(* Logix 5000 project; controller AdvManLab vendor 1 type 14 code 158 rev 28.12; software revision 28.01; part 11 of 13 *)
(* tags used below, declared in another part *)
   RFID_Address : DINT;
   RFID_Length : DINT;
   RFID_Read_1 : BOOL;
   RFID_Read_3 : BOOL;
   RFID_Read_5 : BOOL;
   RFID_Read_Byte_Start_1 : BOOL;
   RFID_Read_Byte_Start_3 : BOOL;
   RFID_Read_Byte_Start_5 : BOOL;
   RFID_Read_InProgress_1 : BOOL;
   RFID_Read_InProgress_3 : BOOL;
   RFID_Read_InProgress_5 : BOOL;
   ABB_Loop_Conv_ES_Ch1 : BOOL;   // Cell 3 Conveyor Pull Cord / E-Stop Ch1
   ABB_Loop_Conv_ES_Ch2 : BOOL;   // Cell 3 Conveyor Pull Cord / E-Stop Ch2
   ABB_Loop_Conv_Safety_OK : BOOL;
   ABBLoopPullCordES : EMERGENCY_STOP;   // EStop / Cable On ABB Loop
   ABBLoopSTO_O1 : BOOL;
   ABBLoopSTO_O2 : BOOL;
   ASynch : BOOL;
   AutoProgStart : TIMER;
   C1_Robot_ES_OK : BOOL;
   C1_Robot_Gates_OK : BOOL;
   C1S : Fanuc_Cell_Safe;
   C2_Robot_ES_OK : BOOL;
   C2_Robot_Gates_OK : BOOL;
   C2S : Fanuc_Cell_Safe;
   C3_Robot_ES_OK : BOOL;
   C3_Robot_Gates_OK : BOOL;
   C3S : ABB_Cell_Safe;
   Cell1EntryLC : LIGHT_CURTAIN;   // Cell 1 Conveyor Entry Light Screen
   Cell1EntryLCMute : MUTING_TWO_SENSOR_SYM;   // Celll 1 Entry LC Muting
   Cell1ExitLC : LIGHT_CURTAIN;   // Cell 1 Conveyor Exit Light Screen
   Cell1ExitLCMute : MUTING_TWO_SENSOR_SYM;   // Celll 1 Exit LC Muting
   Cell1GateSW : REDUNDANT_INPUT;   // Cell 1 Entry Gate Switch
   Cell2EntryLC : LIGHT_CURTAIN;   // Cell 2 Conveyor Entry Light Screen
   Cell2EntryLCMute : MUTING_TWO_SENSOR_SYM;   // Celll 2 Entry LC Muting
   Cell2ExitLC : LIGHT_CURTAIN;   // Cell 2 Conveyor Exit Light Screen
   Cell2ExitLCMute : MUTING_TWO_SENSOR_SYM;   // Celll 2 Exit LC Muting
   Cell2GateSW : REDUNDANT_INPUT;   // Cell 2 Entry Gate Switch
   Cell3EntryLC : LIGHT_CURTAIN;   // Cell 3 Conveyor Entry Light Screen
   Cell3EntryLCMute : MUTING_TWO_SENSOR_SYM;   // Celll 3 Entry LC Muting
   Cell3ExitLC : LIGHT_CURTAIN;   // Cell 3 Conveyor Exit Light Screen
   Cell3ExitLCMute : MUTING_TWO_SENSOR_SYM;   // Celll 3 Exit LC Muting
   Cell3GateSW : REDUNDANT_INPUT;   // Cell 3 Entry Gate Switch
   Cell_1 : Fanuc_Cell;
   Cell_2 : Fanuc_Cell;
   CircuitResetSafe : BOOL;   // Signal to Reset Circuits
   CNC1_Door : REDUNDANT_INPUT;   // CNC1 Door Switch
   CNC1_EStop : EMERGENCY_STOP;
   CNC1_LC : LIGHT_CURTAIN;   // CNC1 to Cell 1 Light Screen
   CNC2_Door : REDUNDANT_INPUT;   // CNC2 Door Switch
   CNC2_EStop : EMERGENCY_STOP;
   CNC2_LC : LIGHT_CURTAIN;   // CNC2 to Cell 1 Light Screen
   CNC3_Door : REDUNDANT_INPUT;   // CNC3 Door Switch
   CNC3_EStop : EMERGENCY_STOP;
   CNC3_LC : LIGHT_CURTAIN;   // CNC3 to Cell 2 Light Screen
   CNC4_Door : REDUNDANT_INPUT;   // CNC4 Door Switch
   CNC4_EStop : EMERGENCY_STOP;
   CNC4_LC : LIGHT_CURTAIN;   // CNC4 to Cell 2 Light Screen
   ContinuousRunCase : BOOL;
   Dry_Cycle : BOOL;
   Fanuc_Loop_Conv_ES_Ch1 : BOOL;   // Cell 1/2 Conveyor Pull Cord / E-Stop Ch1
   Fanuc_Loop_Conv_ES_Ch2 : BOOL;   // Cell 1/2 Conveyor Pull Cord / E-Stop Ch2
   Fanuc_Loop_Conv_Safety_OK : BOOL;
   Fanuc_Loop_Speed : DINT;
   FanucLoopPullCordES : EMERGENCY_STOP;   // EStop / Cable On Fanuc Loop
   FanucLoopSTO_O1 : BOOL;
   FanucLoopSTO_O2 : BOOL;
   FanucLoopVFD : PF525_Faceplate_AOI;
   FaultReset : BOOL;
   FaultResetSafe : BOOL;
   MainPnlES : EMERGENCY_STOP;   // EStop on Main Panel
   MainPnlESCH1 : BOOL;   // Main Panel E-Stop Button CH1
   MainPnlESCH2 : BOOL;   // Main Panel E-Stop Button CH2
   Mode_Auto : BOOL;
   Mode_Manual : BOOL;
   PaletClearPreset : DINT[8];
   PF525_FaultCodeList : P_DescList[61];   // PowerFlex 525 VFD Fault Codes and Descriptions
   R1J_Write_Inprogress : BOOL;
   RelC1HoldBack : TIMER;
   RelC1RobotStop : TIMER;
   RelC2HoldBack : TIMER;
   RelC2RobotStop : TIMER;
   RFID_ReadData1 : SINT;
   RFID_ReadData1p : SINT;
   RFID_ReadData1process : DINT;
   RFID_ReadData1processtime : DINT;
   RFID_ReadData1timer : SINT[4];
   RFID_ReadData3 : SINT;
   RFID_ReadData3p : DINT;
   RFID_ReadData3process : DINT;
   RFID_ReadData3processtime : DINT;
   RFID_ReadData3timer : SINT[4];
   RFID_ReadData5 : SINT;
   RFID_ReadData5p : DINT;
   RFID_ReadData5process : DINT;
   RFID_ReadData5processtime : DINT;
   RFID_ReadData5timer : SINT[4];
   RFID_Write_1 : BOOL;
   RFID_Write_3 : BOOL;
   RFID_Write_5 : BOOL;
   RFIDTP1 : ALIAS FOR RFID_N054:I.Channel[0].TagPresent;   // RFID Tag at Cell 1 Stop
   RFIDTP3 : ALIAS FOR RFID_N055:I.Channel[0].TagPresent;   // RFID Tag at Cell 2 Stop
   RFIDTP5 : ALIAS FOR RFID_N056:I.Channel[0].TagPresent;   // RFID Tag at Cell 3 Stop
   RunABBLoopatSpeed : BOOL;
   RunASynchCase : BOOL;
   RunCont : BOOL;
   RungCommentS : BOOL;
   RunSynch : BOOL;
   RunSynchCase : BOOL;
   SC105 : P_PF52x;   // Pump 105 Motor (PowerFlex 525 drive)
   so_AcceptMSG00 : MESSAGE;
   so_CreateInstance : DINT;
   so_CreateMSG00 : MESSAGE;
   so_CreateParams : AcceptResponse;
   so_OpenMSG00 : MESSAGE;
   Timer_RFID1 : TIMER;
   Timer_RFID3 : TIMER;
   Timer_RFID5 : TIMER;
   VFDFanucLoop_I : P_PF52x_Inp;
   VFDFanucLoop_O : P_PF52x_Out;
(* MainProgram, continued *)

ROUTINE RFID_HMI   (* ladder *)
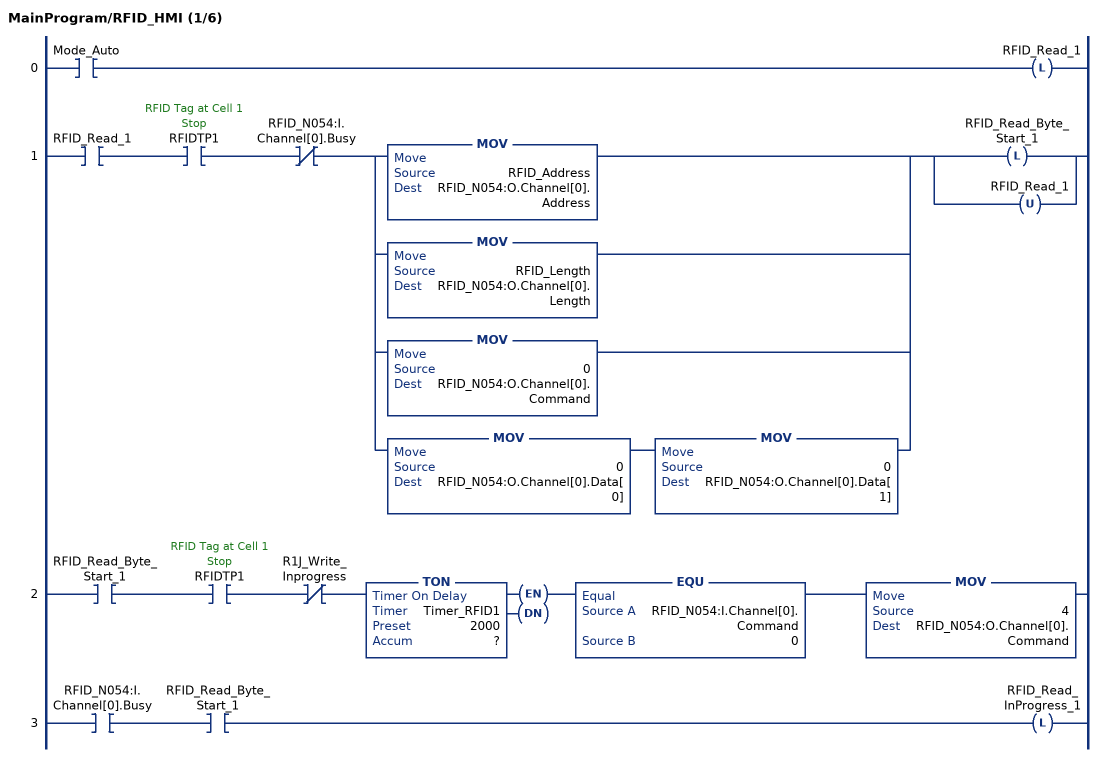
   0: XIC(Mode_Auto)OTL(RFID_Read_1);
   1: XIC(RFID_Read_1)XIC(RFIDTP1)XIO(RFID_N054:I.Channel[0].Busy)[MOV(RFID_Address,RFID_N054:O.Channel[0].Address) ,MOV(RFID_Length,RFID_N054:O.Channel[0].Length) ,[MOV(0,RFID_N054:O.Channel[0].Command) ,MOV(0,RFID_N054:O.Channel[0].Data[0]) MOV(0,RFID_N054:O.Channel[0].Data[1]) ] ][OTL(RFID_Read_Byte_Start_1) ,OTU(RFID_Read_1) ];
   2: XIC(RFID_Read_Byte_Start_1)XIC(RFIDTP1)XIO(R1J_Write_Inprogress)TON(Timer_RFID1,?,?)EQU(RFID_N054:I.Channel[0].Command,0)MOV(4,RFID_N054:O.Channel[0].Command);
   3: XIC(RFID_N054:I.Channel[0].Busy)XIC(RFID_Read_Byte_Start_1)OTL(RFID_Read_InProgress_1);
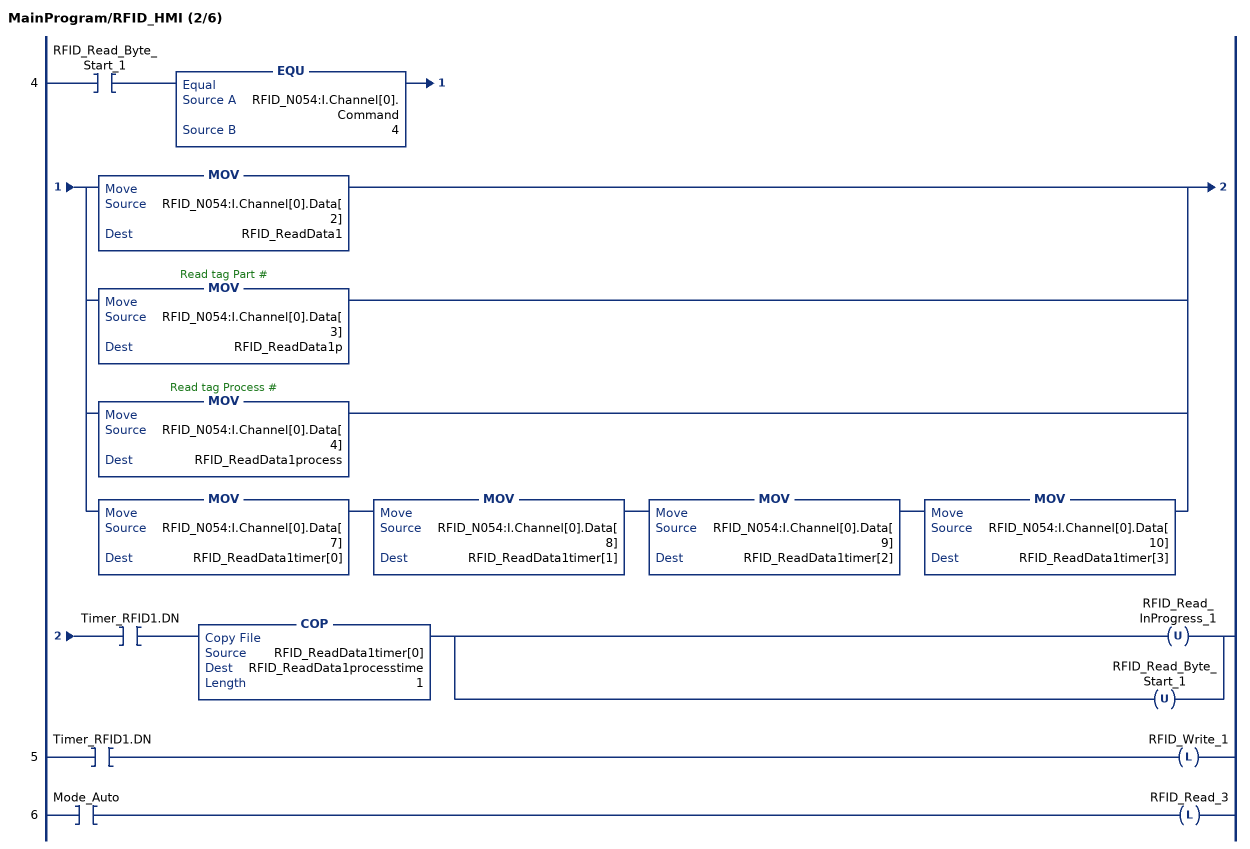
   4: XIC(RFID_Read_Byte_Start_1)EQU(RFID_N054:I.Channel[0].Command,4)[MOV(RFID_N054:I.Channel[0].Data[2],RFID_ReadData1) ,[MOV(RFID_N054:I.Channel[0].Data[3],RFID_ReadData1p) ,[MOV(RFID_N054:I.Channel[0].Data[4],RFID_ReadData1process) ,MOV(RFID_N054:I.Channel[0].Data[7],RFID_ReadData1timer[0]) MOV(RFID_N054:I.Channel[0].Data[8],RFID_ReadData1timer[1]) MOV(RFID_N054:I.Channel[0].Data[9],RFID_ReadData1timer[2]) MOV(RFID_N054:I.Channel[0].Data[10],RFID_ReadData1timer[3]) ] ] ]XIC(Timer_RFID1.DN)COP(RFID_ReadData1timer[0],RFID_ReadData1processtime,1)[OTU(RFID_Read_InProgress_1) ,OTU(RFID_Read_Byte_Start_1) ];
   5: XIC(Timer_RFID1.DN)OTL(RFID_Write_1);
   6: XIC(Mode_Auto)OTL(RFID_Read_3);
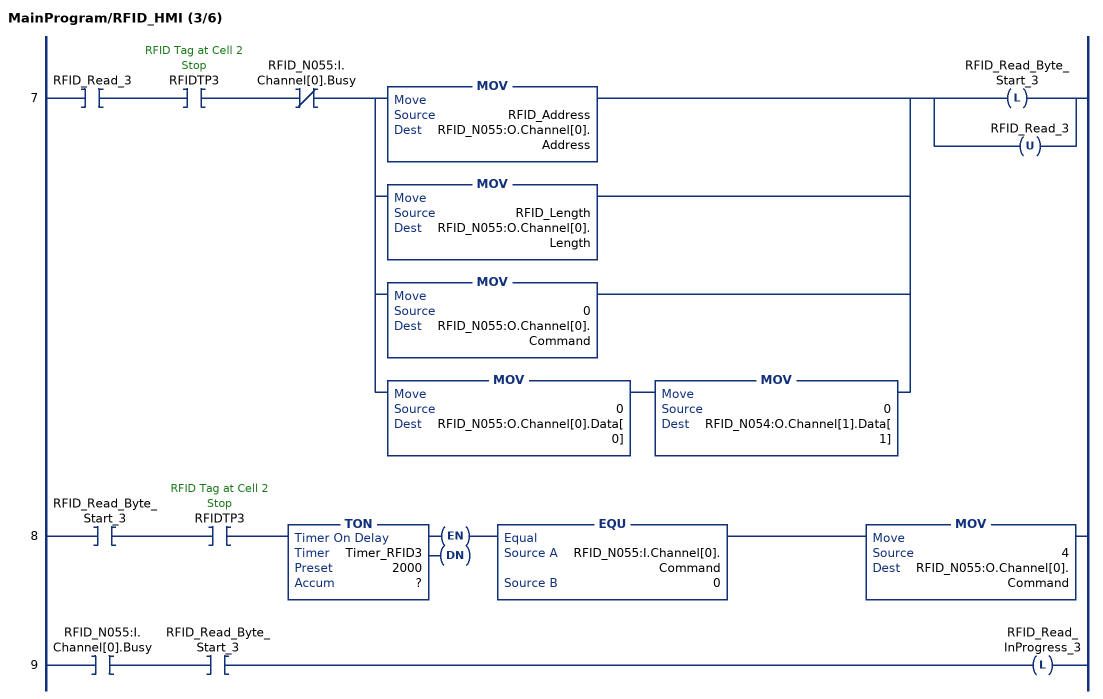
   7: XIC(RFID_Read_3)XIC(RFIDTP3)XIO(RFID_N055:I.Channel[0].Busy)[MOV(RFID_Address,RFID_N055:O.Channel[0].Address) ,MOV(RFID_Length,RFID_N055:O.Channel[0].Length) ,[MOV(0,RFID_N055:O.Channel[0].Command) ,MOV(0,RFID_N055:O.Channel[0].Data[0]) MOV(0,RFID_N054:O.Channel[1].Data[1]) ] ][OTL(RFID_Read_Byte_Start_3) ,OTU(RFID_Read_3) ];
   8: XIC(RFID_Read_Byte_Start_3)XIC(RFIDTP3)TON(Timer_RFID3,?,?)EQU(RFID_N055:I.Channel[0].Command,0)MOV(4,RFID_N055:O.Channel[0].Command);
   9: XIC(RFID_N055:I.Channel[0].Busy)XIC(RFID_Read_Byte_Start_3)OTL(RFID_Read_InProgress_3);
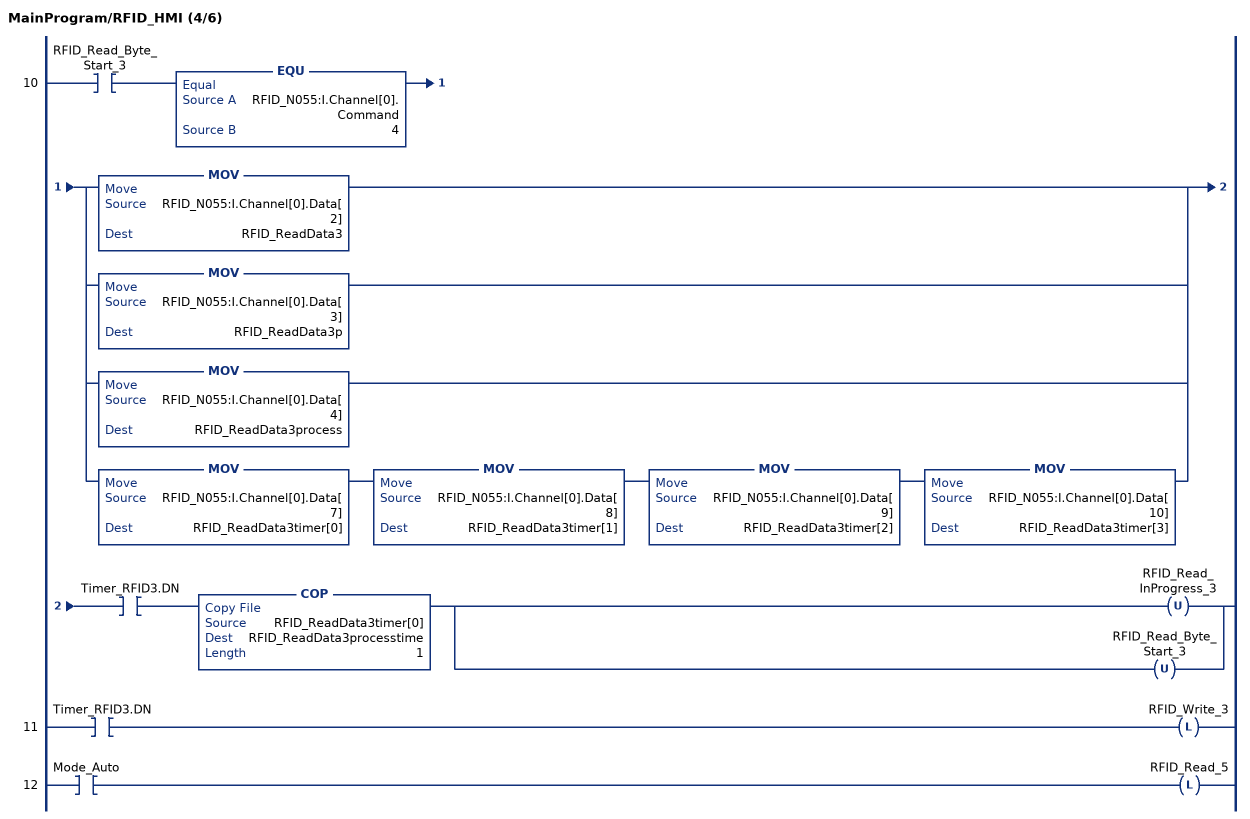
   10: XIC(RFID_Read_Byte_Start_3)EQU(RFID_N055:I.Channel[0].Command,4)[MOV(RFID_N055:I.Channel[0].Data[2],RFID_ReadData3) ,[MOV(RFID_N055:I.Channel[0].Data[3],RFID_ReadData3p) ,[MOV(RFID_N055:I.Channel[0].Data[4],RFID_ReadData3process) ,MOV(RFID_N055:I.Channel[0].Data[7],RFID_ReadData3timer[0]) MOV(RFID_N055:I.Channel[0].Data[8],RFID_ReadData3timer[1]) MOV(RFID_N055:I.Channel[0].Data[9],RFID_ReadData3timer[2]) MOV(RFID_N055:I.Channel[0].Data[10],RFID_ReadData3timer[3]) ] ] ]XIC(Timer_RFID3.DN)COP(RFID_ReadData3timer[0],RFID_ReadData3processtime,1)[OTU(RFID_Read_InProgress_3) ,OTU(RFID_Read_Byte_Start_3) ];
   11: XIC(Timer_RFID3.DN)OTL(RFID_Write_3);
   12: XIC(Mode_Auto)OTL(RFID_Read_5);
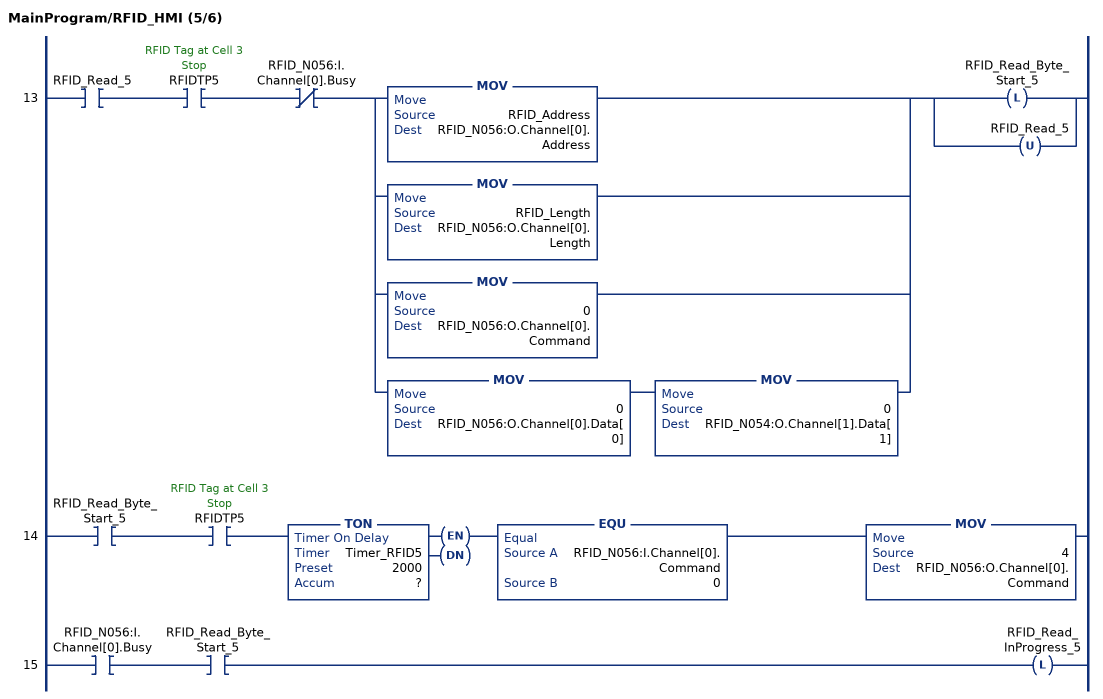
   13: XIC(RFID_Read_5)XIC(RFIDTP5)XIO(RFID_N056:I.Channel[0].Busy)[MOV(RFID_Address,RFID_N056:O.Channel[0].Address) ,MOV(RFID_Length,RFID_N056:O.Channel[0].Length) ,[MOV(0,RFID_N056:O.Channel[0].Command) ,MOV(0,RFID_N056:O.Channel[0].Data[0]) MOV(0,RFID_N054:O.Channel[1].Data[1]) ] ][OTL(RFID_Read_Byte_Start_5) ,OTU(RFID_Read_5) ];
   14: XIC(RFID_Read_Byte_Start_5)XIC(RFIDTP5)TON(Timer_RFID5,?,?)EQU(RFID_N056:I.Channel[0].Command,0)MOV(4,RFID_N056:O.Channel[0].Command);
   15: XIC(RFID_N056:I.Channel[0].Busy)XIC(RFID_Read_Byte_Start_5)OTL(RFID_Read_InProgress_5);
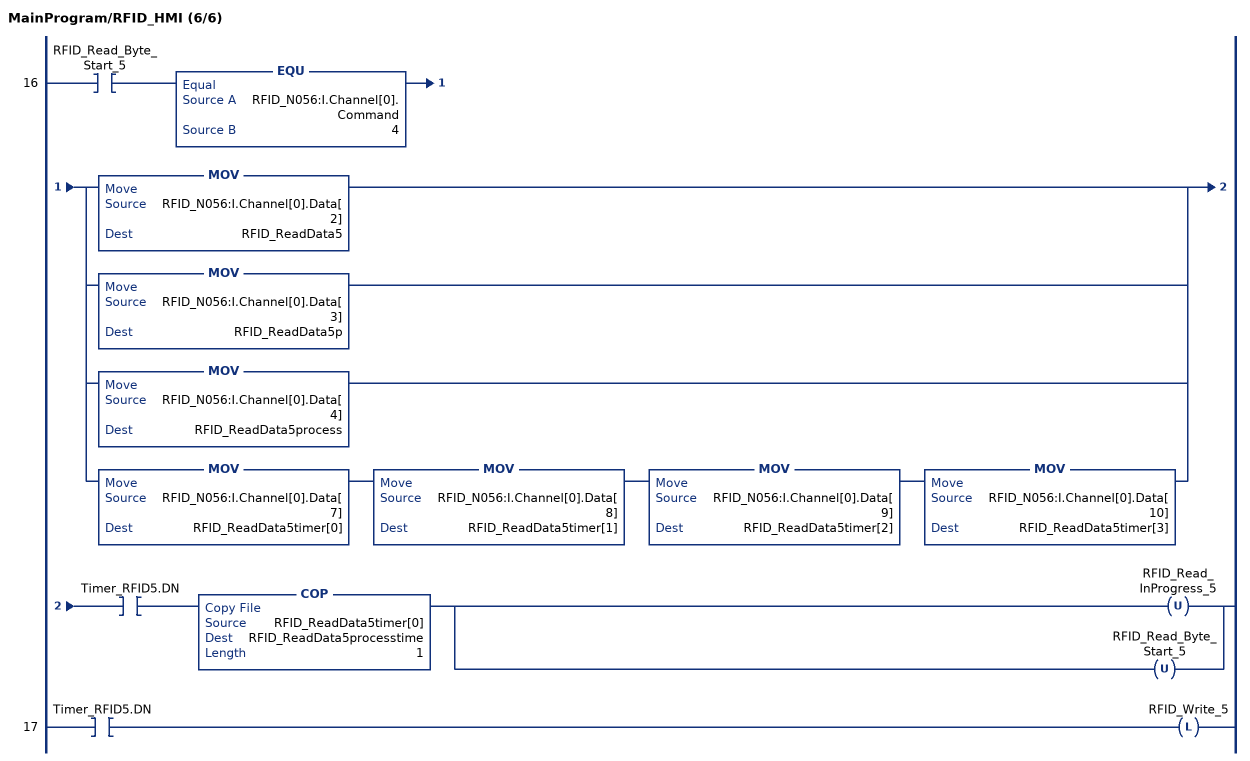
   16: XIC(RFID_Read_Byte_Start_5)EQU(RFID_N056:I.Channel[0].Command,4)[MOV(RFID_N056:I.Channel[0].Data[2],RFID_ReadData5) ,[MOV(RFID_N056:I.Channel[0].Data[3],RFID_ReadData5p) ,[MOV(RFID_N056:I.Channel[0].Data[4],RFID_ReadData5process) ,MOV(RFID_N056:I.Channel[0].Data[7],RFID_ReadData5timer[0]) MOV(RFID_N056:I.Channel[0].Data[8],RFID_ReadData5timer[1]) MOV(RFID_N056:I.Channel[0].Data[9],RFID_ReadData5timer[2]) MOV(RFID_N056:I.Channel[0].Data[10],RFID_ReadData5timer[3]) ] ] ]XIC(Timer_RFID5.DN)COP(RFID_ReadData5timer[0],RFID_ReadData5processtime,1)[OTU(RFID_Read_InProgress_5) ,OTU(RFID_Read_Byte_Start_5) ];
   17: XIC(Timer_RFID5.DN)OTL(RFID_Write_5);
END_ROUTINE

ROUTINE System   (* ladder *)
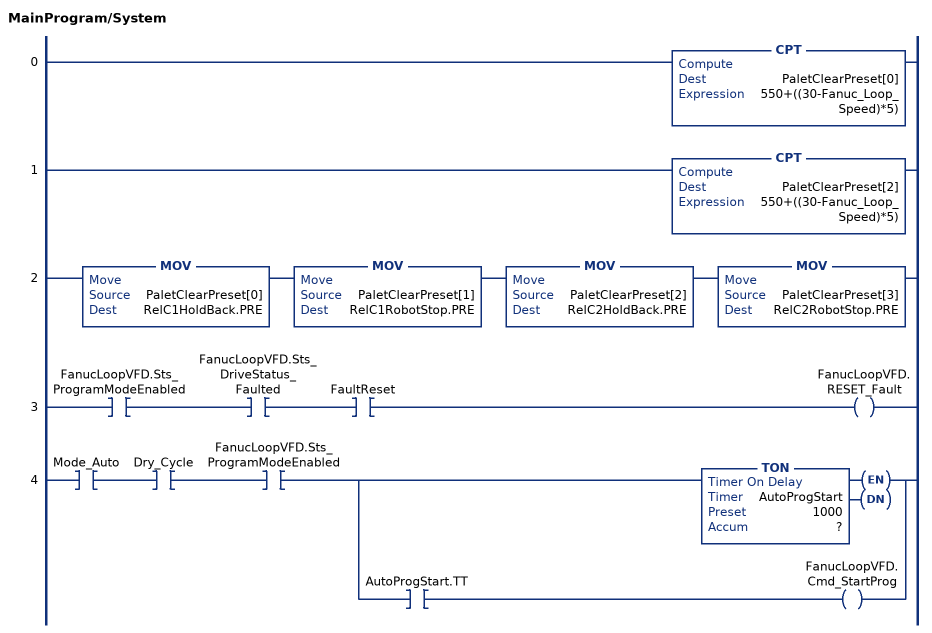
   0: CPT(PaletClearPreset[0],550+((30-Fanuc_Loop_Speed)*5));
   1: CPT(PaletClearPreset[2],550+((30-Fanuc_Loop_Speed)*5));
   2: MOV(PaletClearPreset[0],RelC1HoldBack.PRE)MOV(PaletClearPreset[1],RelC1RobotStop.PRE)MOV(PaletClearPreset[2],RelC2HoldBack.PRE)MOV(PaletClearPreset[3],RelC2RobotStop.PRE);
   3: XIC(FanucLoopVFD.Sts_ProgramModeEnabled)XIC(FanucLoopVFD.Sts_DriveStatus_Faulted)XIC(FaultReset)OTE(FanucLoopVFD.RESET_Fault);
   4: XIC(Mode_Auto)XIC(Dry_Cycle)XIC(FanucLoopVFD.Sts_ProgramModeEnabled)[TON(AutoProgStart,?,?) ,XIC(AutoProgStart.TT) OTE(FanucLoopVFD.Cmd_StartProg) ];
END_ROUTINE

ROUTINE Unused_PF52x   (* ladder *)
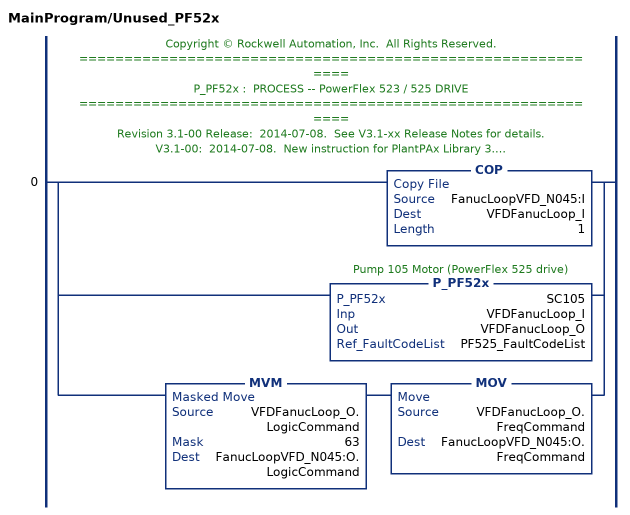
   // Copyright © Rockwell Automation, Inc.  All Rights Reserved.
   // ============================================================
   // P_PF52x :  PROCESS -- PowerFlex 523 / 525 DRIVE
   // ============================================================
   // Revision 3.1-00 Release:  2014-07-08.  See V3.1-xx Release Notes for details.
   // V3.1-00:  2014-07-08.  New instruction for PlantPAx Library 3.1
   // ============================================================
   // This Instruction controls and monitors a PowerFlex 523 Variable-Frequency Drive with
   // optional EtherNet/IP Interface, or a PowerFlex 525 Variable-Frequency
   // Drive with embedded or optional add-on EtherNet/IP Interface.
   // ============================================================
   // REQUIRED DRIVE CONFIGURATION
   // ============================================================
   // Be certain to set up the drive Datalinks as follows!
   // 'User Choice' Datalinks are not used by this AOI and
   // may be left unused or set up for your application.
   // INPUT ASSEMBLY:
   // Drive Status (standard)
   // Output Frequency (standard)
   // 1. Fault 1 Code (Par 007)
   // 2. Output Current (Par 003)
   // 3. Output Power (Par 017)
   // 4. User choice
   // OUTPUT ASSEMBLY:
   // Drive Logic Comnmand (standard)
   // Frequency Command (Speed Reference) (standard)
   // All 4 output datalinks are user choice.
   // ============================================================
   // Create a Tag of type P_PF52x_Inp, and create a Tag of type P_PF52x_Out
   // to buffer the starter's Input and Output data.  Then add these Tags in the Input
   // and Output parameters of the P_PF52x instruction instance and replace
   // operands in the "COP" and "MVM"/"MOV" instructions as described below.
   // In these examples, the names given to various tags are as follows:
   // *  The backing tag for the P_PF52x AOI is "SC105".
   // *  The Input buffer tag (of type P_PF52x_Inp) is "SC105_I".
   // *  The Output buffer tag (of type P_PF52x_Out) is "SC105_O".
   // *  The PowerFlex 525 drive in the I/O tree of the controller
   // organizer is "SC105_Drive".
   // *  Given that name, the drive's Input Assembly is "SC105_Drive:I"
   // and its Output Assembly is "SC105_Drive:O".
   // 1.  In the COP, replace the Source operand with the actual
   // Input assembly from the starter, and replace the Destination
   // operand with the input buffer tag of type P_PF52x_Inp you created,
   // for example:
   // COP
   // SC105_Drive:I
   // SC105_I
   // Len=1
   // 2.  In the AOI instance, put the buffer tags in the InOut parameters,
   // for example:
   // Inp  is  SC105_I
   // Out  is  SC105_O
   // 2.  In the MVM, replace the Source operand with the LogicCommand
   // element of the Tag of type P_PF52x_Out you created, and replace
   // the Destination operand with the LogicCommand element of the
   // actual Output Assembly going to the drive, for example:
   // MVM
   // SC105_O.LogicCommand
   // 2#0000_0000_0011_1111
   // SC105_Drive:O.LogicCommand
   // 3.  In the MOV, replace the Source operand with the Reference
   // element of the Tag of type P_PF52x_Out which you created, and
   // replace the Destination operand with the Reference element
   // of the actual Output Assembly going to the drive, for example:
   // MOV
   // SC105_O.FreqCommand
   // SC105_Drive:O.FreqCommand
   0: [COP(FanucLoopVFD_N045:I,VFDFanucLoop_I,1) ,P_PF52x(SC105,VFDFanucLoop_I,VFDFanucLoop_O,PF525_FaultCodeList) ,MVM(VFDFanucLoop_O.LogicCommand,63,FanucLoopVFD_N045:O.LogicCommand) MOV(VFDFanucLoop_O.FreqCommand,FanucLoopVFD_N045:O.FreqCommand) ];
END_ROUTINE

ROUTINE Unused_Socket_Test   (* ladder *)
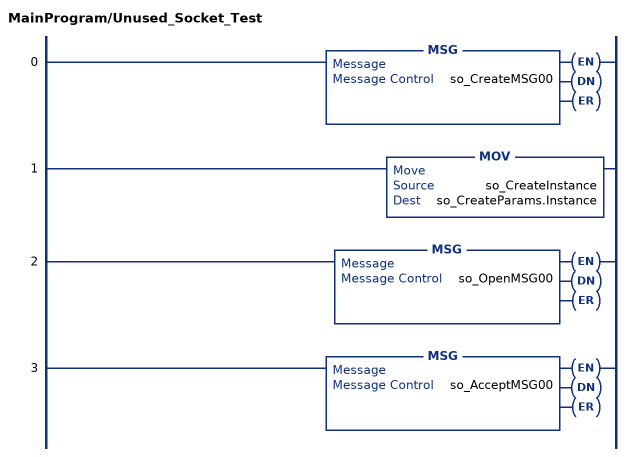
   0: MSG(so_CreateMSG00);
   1: MOV(so_CreateInstance,so_CreateParams.Instance);
   2: MSG(so_OpenMSG00);
   3: MSG(so_AcceptMSG00);
END_ROUTINE

ROUTINE Unused_Vernnaliz   (* ladder *)
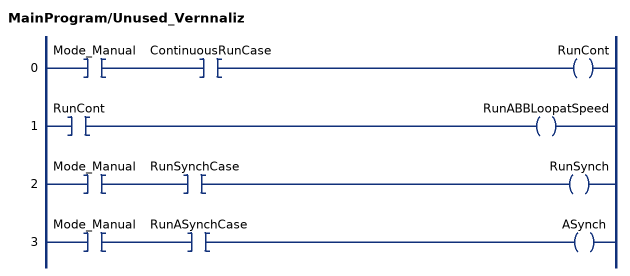
   0: XIC(Mode_Manual)XIC(ContinuousRunCase)OTE(RunCont);
   1: XIC(RunCont)OTE(RunABBLoopatSpeed);
   2: XIC(Mode_Manual)XIC(RunSynchCase)OTE(RunSynch);
   3: XIC(Mode_Manual)XIC(RunASynchCase)OTE(ASynch);
END_ROUTINE
END_PROGRAM

PROGRAM SafetyProgram   (* main routine MainRoutine, safety *)

ROUTINE Cell_1   (* ladder *)
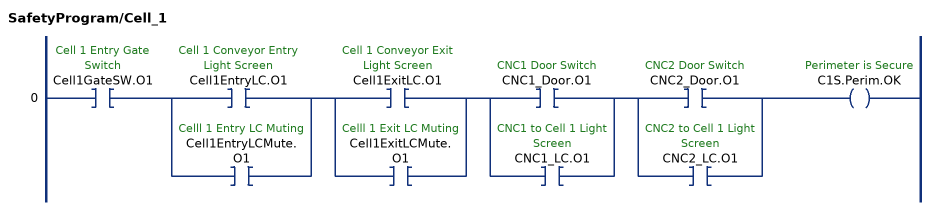
   0: XIC(Cell1GateSW.O1)[XIC(Cell1EntryLC.O1) ,XIC(Cell1EntryLCMute.O1) ][XIC(Cell1ExitLC.O1) ,XIC(Cell1ExitLCMute.O1) ][XIC(CNC1_Door.O1) ,XIC(CNC1_LC.O1) ][XIC(CNC2_Door.O1) ,XIC(CNC2_LC.O1) ]OTE(C1S.Perim.OK);
END_ROUTINE

ROUTINE Cell_1_2_VFD   (* ladder *)
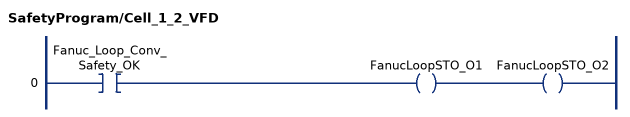
   0: XIC(Fanuc_Loop_Conv_Safety_OK)OTE(FanucLoopSTO_O1)OTE(FanucLoopSTO_O2);
END_ROUTINE

ROUTINE Cell_2   (* ladder *)
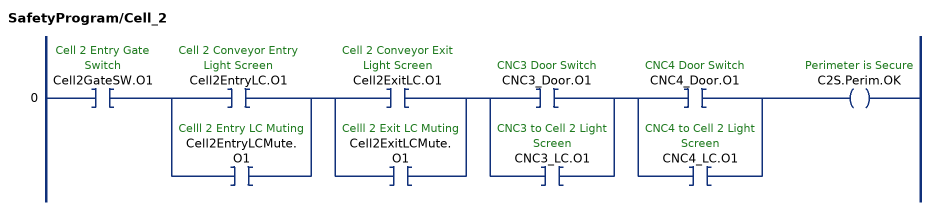
   0: XIC(Cell2GateSW.O1)[XIC(Cell2EntryLC.O1) ,XIC(Cell2EntryLCMute.O1) ][XIC(Cell2ExitLC.O1) ,XIC(Cell2ExitLCMute.O1) ][XIC(CNC3_Door.O1) ,XIC(CNC3_LC.O1) ][XIC(CNC4_Door.O1) ,XIC(CNC4_LC.O1) ]OTE(C2S.Perim.OK);
END_ROUTINE

ROUTINE Cell_3   (* ladder *)
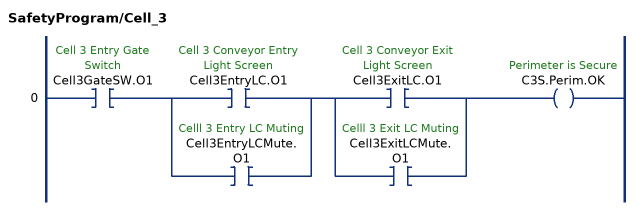
   0: XIC(Cell3GateSW.O1)[XIC(Cell3EntryLC.O1) ,XIC(Cell3EntryLCMute.O1) ][XIC(Cell3ExitLC.O1) ,XIC(Cell3ExitLCMute.O1) ]OTE(C3S.Perim.OK);
END_ROUTINE

ROUTINE Cell_3_VFD   (* ladder *)
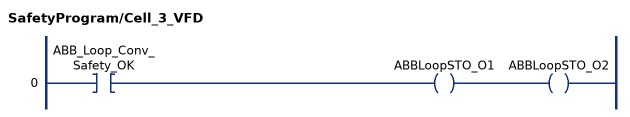
   0: XIC(ABB_Loop_Conv_Safety_OK)OTE(ABBLoopSTO_O1)OTE(ABBLoopSTO_O2);
END_ROUTINE

ROUTINE EStopsAndGates   (* ladder *)
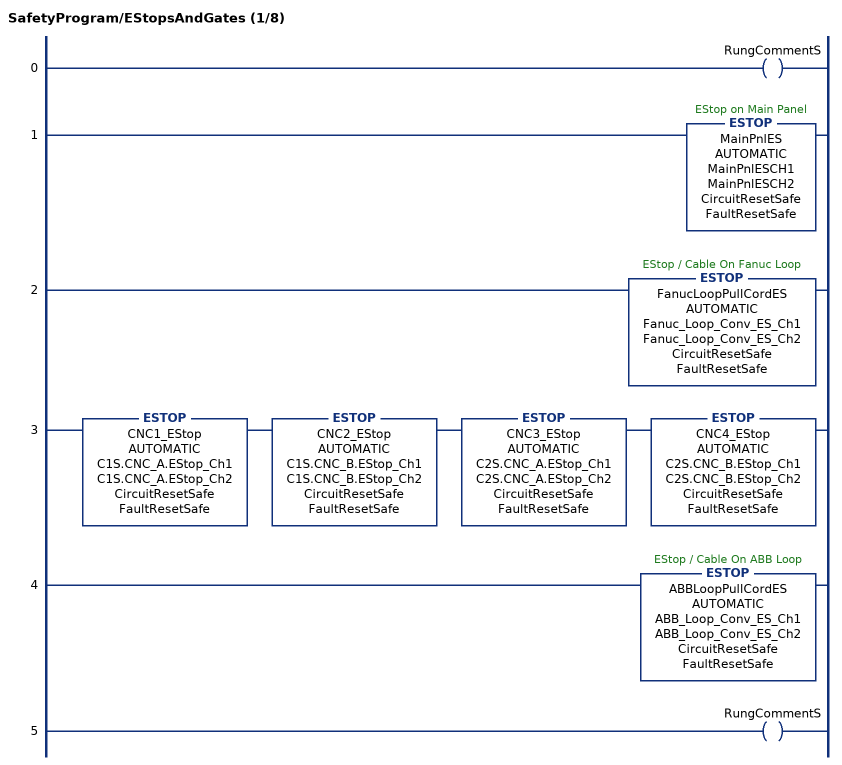
   0: OTE(RungCommentS);
   1: ESTOP(MainPnlES,AUTOMATIC,MainPnlESCH1,MainPnlESCH2,CircuitResetSafe,FaultResetSafe);
   2: ESTOP(FanucLoopPullCordES,AUTOMATIC,Fanuc_Loop_Conv_ES_Ch1,Fanuc_Loop_Conv_ES_Ch2,CircuitResetSafe,FaultResetSafe);
   3: ESTOP(CNC1_EStop,AUTOMATIC,C1S.CNC_A.EStop_Ch1,C1S.CNC_A.EStop_Ch2,CircuitResetSafe,FaultResetSafe)ESTOP(CNC2_EStop,AUTOMATIC,C1S.CNC_B.EStop_Ch1,C1S.CNC_B.EStop_Ch2,CircuitResetSafe,FaultResetSafe)ESTOP(CNC3_EStop,AUTOMATIC,C2S.CNC_A.EStop_Ch1,C2S.CNC_A.EStop_Ch2,CircuitResetSafe,FaultResetSafe)ESTOP(CNC4_EStop,AUTOMATIC,C2S.CNC_B.EStop_Ch1,C2S.CNC_B.EStop_Ch2,CircuitResetSafe,FaultResetSafe);
   4: ESTOP(ABBLoopPullCordES,AUTOMATIC,ABB_Loop_Conv_ES_Ch1,ABB_Loop_Conv_ES_Ch2,CircuitResetSafe,FaultResetSafe);
   5: OTE(RungCommentS);
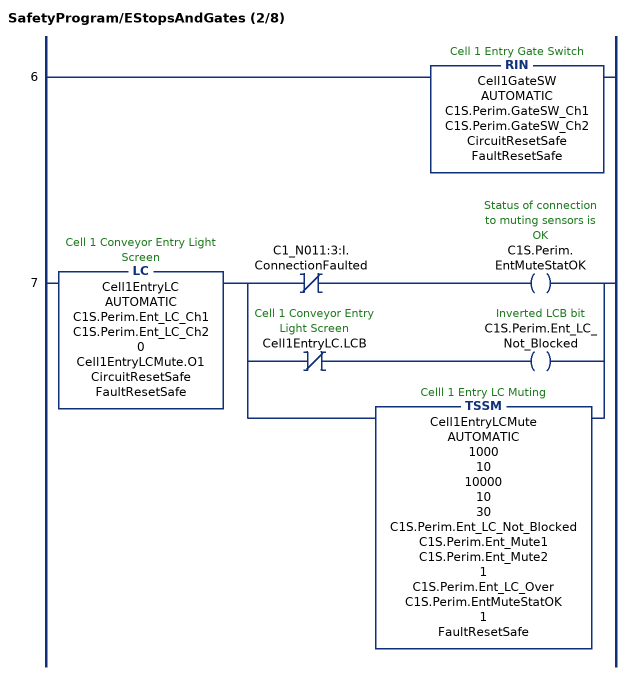
   6: RIN(Cell1GateSW,AUTOMATIC,C1S.Perim.GateSW_Ch1,C1S.Perim.GateSW_Ch2,CircuitResetSafe,FaultResetSafe);
   7: LC(Cell1EntryLC,AUTOMATIC,C1S.Perim.Ent_LC_Ch1,C1S.Perim.Ent_LC_Ch2,0,Cell1EntryLCMute.O1,CircuitResetSafe,FaultResetSafe)[XIO(C1_N011:3:I.ConnectionFaulted) OTE(C1S.Perim.EntMuteStatOK) ,XIO(Cell1EntryLC.LCB) OTE(C1S.Perim.Ent_LC_Not_Blocked) ,TSSM(Cell1EntryLCMute,AUTOMATIC,1000,10,10000,10,30,C1S.Perim.Ent_LC_Not_Blocked,C1S.Perim.Ent_Mute1,C1S.Perim.Ent_Mute2,1,C1S.Perim.Ent_LC_Over,C1S.Perim.EntMuteStatOK,1,FaultResetSafe) ];
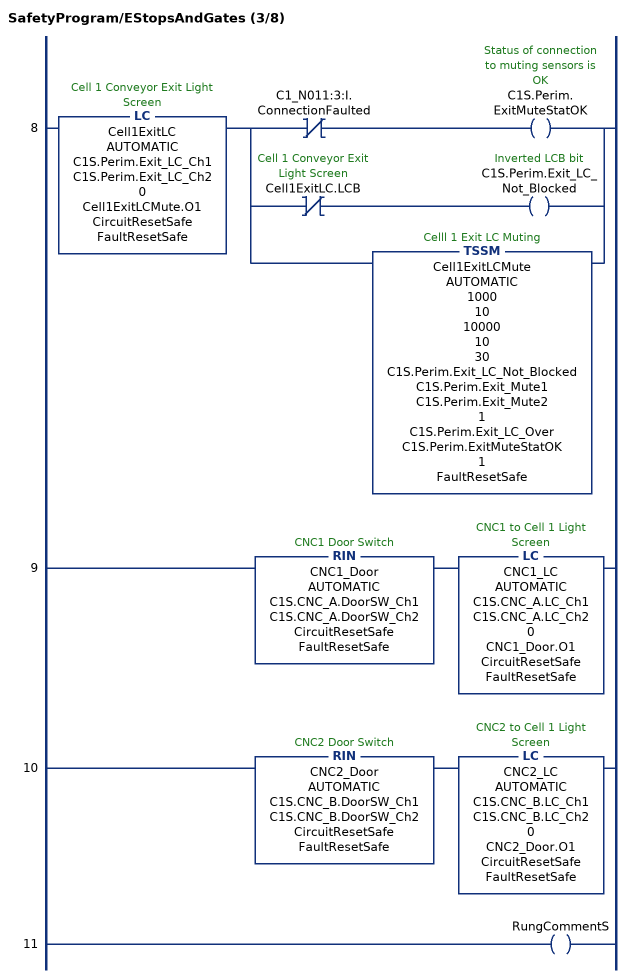
   8: LC(Cell1ExitLC,AUTOMATIC,C1S.Perim.Exit_LC_Ch1,C1S.Perim.Exit_LC_Ch2,0,Cell1ExitLCMute.O1,CircuitResetSafe,FaultResetSafe)[XIO(C1_N011:3:I.ConnectionFaulted) OTE(C1S.Perim.ExitMuteStatOK) ,XIO(Cell1ExitLC.LCB) OTE(C1S.Perim.Exit_LC_Not_Blocked) ,TSSM(Cell1ExitLCMute,AUTOMATIC,1000,10,10000,10,30,C1S.Perim.Exit_LC_Not_Blocked,C1S.Perim.Exit_Mute1,C1S.Perim.Exit_Mute2,1,C1S.Perim.Exit_LC_Over,C1S.Perim.ExitMuteStatOK,1,FaultResetSafe) ];
   9: RIN(CNC1_Door,AUTOMATIC,C1S.CNC_A.DoorSW_Ch1,C1S.CNC_A.DoorSW_Ch2,CircuitResetSafe,FaultResetSafe)LC(CNC1_LC,AUTOMATIC,C1S.CNC_A.LC_Ch1,C1S.CNC_A.LC_Ch2,0,CNC1_Door.O1,CircuitResetSafe,FaultResetSafe);
   10: RIN(CNC2_Door,AUTOMATIC,C1S.CNC_B.DoorSW_Ch1,C1S.CNC_B.DoorSW_Ch2,CircuitResetSafe,FaultResetSafe)LC(CNC2_LC,AUTOMATIC,C1S.CNC_B.LC_Ch1,C1S.CNC_B.LC_Ch2,0,CNC2_Door.O1,CircuitResetSafe,FaultResetSafe);
   11: OTE(RungCommentS);
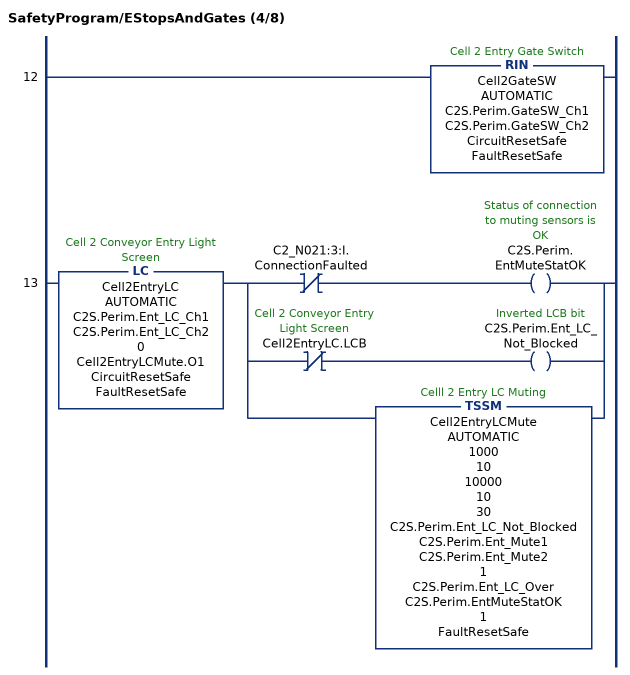
   12: RIN(Cell2GateSW,AUTOMATIC,C2S.Perim.GateSW_Ch1,C2S.Perim.GateSW_Ch2,CircuitResetSafe,FaultResetSafe);
   13: LC(Cell2EntryLC,AUTOMATIC,C2S.Perim.Ent_LC_Ch1,C2S.Perim.Ent_LC_Ch2,0,Cell2EntryLCMute.O1,CircuitResetSafe,FaultResetSafe)[XIO(C2_N021:3:I.ConnectionFaulted) OTE(C2S.Perim.EntMuteStatOK) ,XIO(Cell2EntryLC.LCB) OTE(C2S.Perim.Ent_LC_Not_Blocked) ,TSSM(Cell2EntryLCMute,AUTOMATIC,1000,10,10000,10,30,C2S.Perim.Ent_LC_Not_Blocked,C2S.Perim.Ent_Mute1,C2S.Perim.Ent_Mute2,1,C2S.Perim.Ent_LC_Over,C2S.Perim.EntMuteStatOK,1,FaultResetSafe) ];
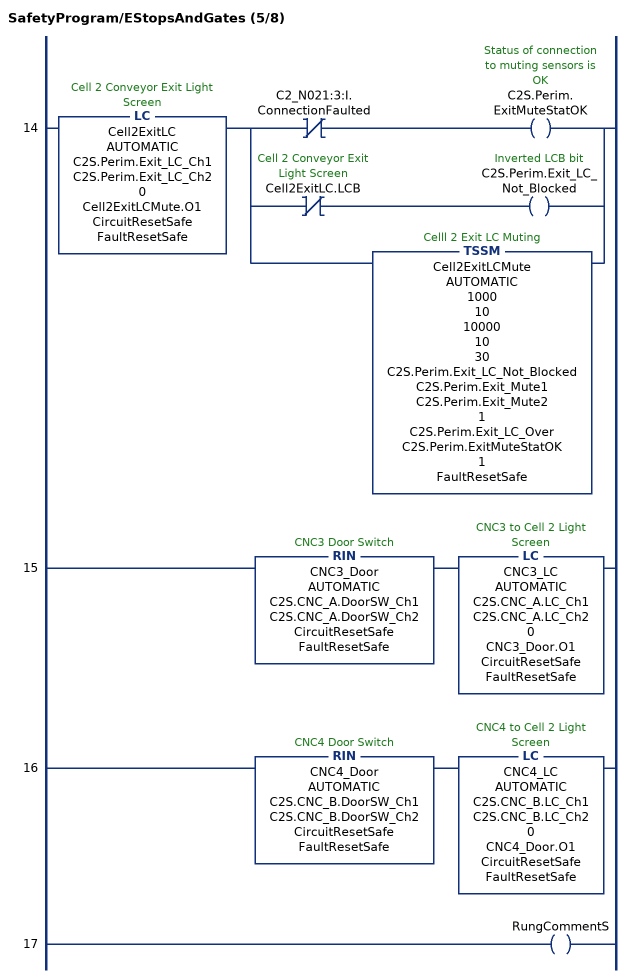
   14: LC(Cell2ExitLC,AUTOMATIC,C2S.Perim.Exit_LC_Ch1,C2S.Perim.Exit_LC_Ch2,0,Cell2ExitLCMute.O1,CircuitResetSafe,FaultResetSafe)[XIO(C2_N021:3:I.ConnectionFaulted) OTE(C2S.Perim.ExitMuteStatOK) ,XIO(Cell2ExitLC.LCB) OTE(C2S.Perim.Exit_LC_Not_Blocked) ,TSSM(Cell2ExitLCMute,AUTOMATIC,1000,10,10000,10,30,C2S.Perim.Exit_LC_Not_Blocked,C2S.Perim.Exit_Mute1,C2S.Perim.Exit_Mute2,1,C2S.Perim.Exit_LC_Over,C2S.Perim.ExitMuteStatOK,1,FaultResetSafe) ];
   15: RIN(CNC3_Door,AUTOMATIC,C2S.CNC_A.DoorSW_Ch1,C2S.CNC_A.DoorSW_Ch2,CircuitResetSafe,FaultResetSafe)LC(CNC3_LC,AUTOMATIC,C2S.CNC_A.LC_Ch1,C2S.CNC_A.LC_Ch2,0,CNC3_Door.O1,CircuitResetSafe,FaultResetSafe);
   16: RIN(CNC4_Door,AUTOMATIC,C2S.CNC_B.DoorSW_Ch1,C2S.CNC_B.DoorSW_Ch2,CircuitResetSafe,FaultResetSafe)LC(CNC4_LC,AUTOMATIC,C2S.CNC_B.LC_Ch1,C2S.CNC_B.LC_Ch2,0,CNC4_Door.O1,CircuitResetSafe,FaultResetSafe);
   17: OTE(RungCommentS);
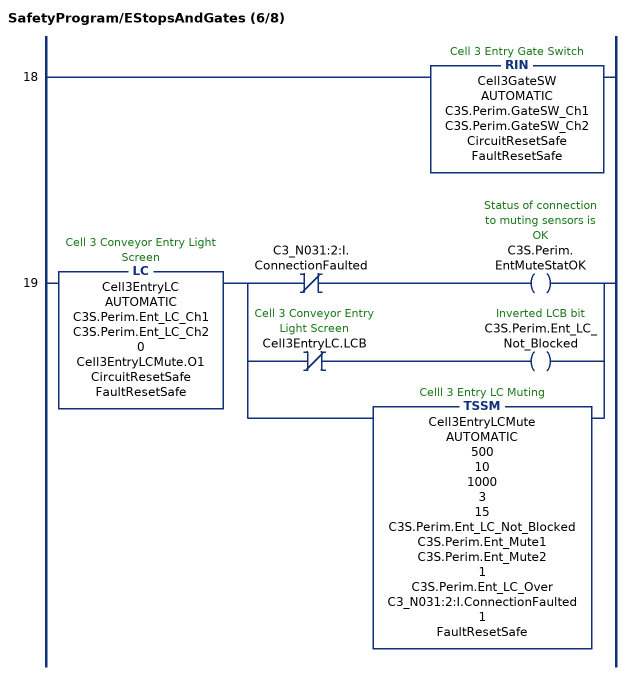
   18: RIN(Cell3GateSW,AUTOMATIC,C3S.Perim.GateSW_Ch1,C3S.Perim.GateSW_Ch2,CircuitResetSafe,FaultResetSafe);
   19: LC(Cell3EntryLC,AUTOMATIC,C3S.Perim.Ent_LC_Ch1,C3S.Perim.Ent_LC_Ch2,0,Cell3EntryLCMute.O1,CircuitResetSafe,FaultResetSafe)[XIO(C3_N031:2:I.ConnectionFaulted) OTE(C3S.Perim.EntMuteStatOK) ,XIO(Cell3EntryLC.LCB) OTE(C3S.Perim.Ent_LC_Not_Blocked) ,TSSM(Cell3EntryLCMute,AUTOMATIC,500,10,1000,3,15,C3S.Perim.Ent_LC_Not_Blocked,C3S.Perim.Ent_Mute1,C3S.Perim.Ent_Mute2,1,C3S.Perim.Ent_LC_Over,C3_N031:2:I.ConnectionFaulted,1,FaultResetSafe) ];
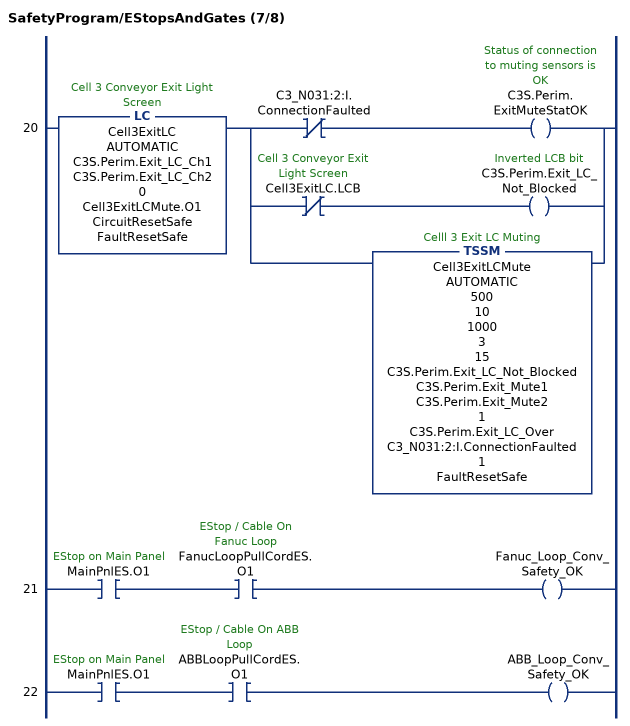
   20: LC(Cell3ExitLC,AUTOMATIC,C3S.Perim.Exit_LC_Ch1,C3S.Perim.Exit_LC_Ch2,0,Cell3ExitLCMute.O1,CircuitResetSafe,FaultResetSafe)[XIO(C3_N031:2:I.ConnectionFaulted) OTE(C3S.Perim.ExitMuteStatOK) ,XIO(Cell3ExitLC.LCB) OTE(C3S.Perim.Exit_LC_Not_Blocked) ,TSSM(Cell3ExitLCMute,AUTOMATIC,500,10,1000,3,15,C3S.Perim.Exit_LC_Not_Blocked,C3S.Perim.Exit_Mute1,C3S.Perim.Exit_Mute2,1,C3S.Perim.Exit_LC_Over,C3_N031:2:I.ConnectionFaulted,1,FaultResetSafe) ];
   21: XIC(MainPnlES.O1)XIC(FanucLoopPullCordES.O1)OTE(Fanuc_Loop_Conv_Safety_OK);
   22: XIC(MainPnlES.O1)XIC(ABBLoopPullCordES.O1)OTE(ABB_Loop_Conv_Safety_OK);
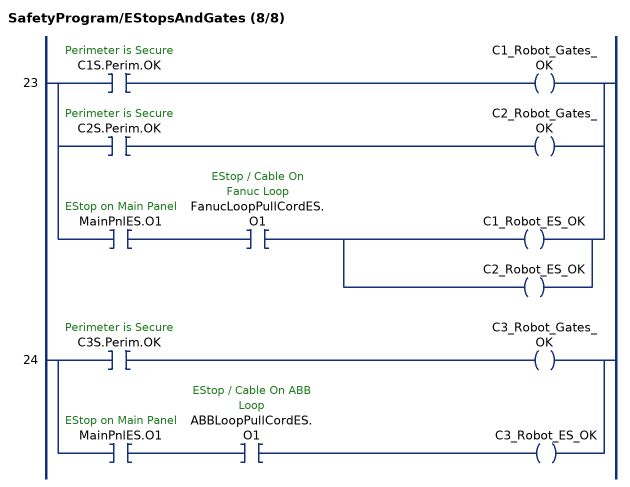
   23: [XIC(C1S.Perim.OK) OTE(C1_Robot_Gates_OK) ,XIC(C2S.Perim.OK) OTE(C2_Robot_Gates_OK) ,XIC(MainPnlES.O1) XIC(FanucLoopPullCordES.O1) [OTE(C1_Robot_ES_OK) ,OTE(C2_Robot_ES_OK) ] ];
   24: [XIC(C3S.Perim.OK) OTE(C3_Robot_Gates_OK) ,XIC(MainPnlES.O1) XIC(ABBLoopPullCordES.O1) OTE(C3_Robot_ES_OK) ];
END_ROUTINE
